// Mitsubishi GX Works2 project: X26   PLC: FX3G

// task Task_01 (event TRUE, interval 0, priority 31): POU_01

PROGRAM POU_01
VAR
  wstep : INT;
  ton1 : TON;
END_VAR
M99 := FALSE AND
M0 AND M2 AND M3 AND 
M4 AND M5 AND M6 AND
Y0 AND Y1 AND Y2 AND
Y3 AND Y4 AND Y5 AND
Y6;

IF M8002 THEN
    wstep := 0;
END_IF;

CASE wstep OF
    0:
        zrst(TRUE, Y0, Y6);        
        ton1(in := FALSE);

        IF M6 THEN
            wstep := 1;
        END_IF;
    1:
        IF M4 THEN
            wstep := 20;
        END_IF;
        IF M5 THEN
            wstep := 40;
        END_IF;

    20:
        Y6 := TRUE;

        IF M0 THEN
            wstep := 21;
        END_IF;
	21:
        Y0 := M2;
        Y1 := M3;
        ton1(in := NOT ton1.q, pt := t#20s);

        IF ton1.q THEN
            Y0 := FALSE;
            Y1 := FALSE;
            wstep := 0;
        END_IF;
      
    40:
        Y5 := TRUE;

        IF M0 THEN
            wstep := 41;
        END_IF;
    41:
        Y2 := TRUE;
        ton1(in := NOT ton1.q, pt := t#5s);

        IF ton1.q THEN
            wstep := 42;
        END_IF;
    42:
        Y2 := FALSE;
        Y3 := TRUE;
        ton1(in := NOT ton1.q, pt := t#5s);

        IF ton1.q THEN
            wstep := 43;
        END_IF;
    43:
        Y3 := FALSE;
        Y4 := TRUE;
        ton1(in := NOT ton1.q, pt := t#10s);
        
        IF ton1.q THEN
            wstep := 0;
        END_IF;
END_CASE;
END_PROGRAM
